// TwinCAT 3 PLC project Untitled1
// ProgramVersion: 3.1.4020.2
// libraries:
//   Tc2_SerialCom, * (Beckhoff Automation GmbH)
//   Tc2_SMS, * (Beckhoff Automation GmbH)
//   Tc2_Standard, * (Beckhoff Automation GmbH)
//   Tc2_System, * (Beckhoff Automation GmbH)
//   Tc2_Utilities, * (Beckhoff Automation GmbH)
//   Tc3_Module, * (Beckhoff Automation GmbH)
//   VisuDialogs, * (System)
// project tree:
//   / FAST_Serial.TcTTO, GlobalTextList.TcGTLO, PlcTask.TcTTO, Visualization Manager.TcVMO (not stored)
//   GVLs/ GVL.TcGVL
//   POUs/ KL6001_Serial.TcPOU, MAIN.TcPOU
//   VISUs/ Visualization.TcVIS
// real-time tasks:
//   TASK PlcTask: cycle T#10ms, priority 20, ADS port 350
//   TASK FAST_Serial: cycle T#1ms, priority 1, ADS port 351
// I/O:
//   DEVICE Device 3 (EtherCAT), AmsNetId 10.123.66.28.4.1
//     Box 1 (BK1150)
// variable links:
//   Untitled1/Untitled1 Instance <-> Device 3 (EtherCAT)/Box 1 (BK1150)
//     PlcTask Inputs/GVL.COMin_EL60xx/D[{0..4}] <-> Term 2 (KL6001-S)/Channel 1/Data In {0..4}  (5 links)
//     PlcTask Inputs/GVL.COMin_EL60xx/Status <-> Term 2 (KL6001-S)/Channel 1/State
//     PlcTask Outputs/GVL.COMout_EL60xx/Ctrl <-> Term 2 (KL6001-S)/Channel 1/Ctrl
//     PlcTask Outputs/GVL.COMout_EL60xx/D[{0..4}] <-> Term 2 (KL6001-S)/Channel 1/Data Out {0..4}  (5 links)

CONFIGURATION Untitled1
    RESOURCE PLC ON TwinCAT3
        TASK FAST_Serial(INTERVAL := T#1ms, PRIORITY := 1);
        TASK PlcTask(INTERVAL := T#10ms, PRIORITY := 20);
        PROGRAM KL6001_Serial WITH FAST_Serial : KL6001_Serial;
        PROGRAM MAIN WITH PlcTask : MAIN;
    END_RESOURCE
END_CONFIGURATION

// ---- GVLs/GVL.TcGVL

VAR_GLOBAL
	COMin_EL60xx	AT %I* 	: KL6InData5B;	(* linked to the EL60xx in the TwinCAT System Manager *)
	COMout_EL60xx	AT %Q*	: KL6OutData5B;	(* linked to the EL60xx in the TwinCAT System Manager *)
	RxBuffer: ComBuffer;						(* Receive data buffer; used with all receive function blocks *)
	TxBuffer: ComBuffer;						(* Transmit data buffer; used with all receive function blocks *)
END_VAR

// ---- POUs/KL6001_Serial.TcPOU
PROGRAM KL6001_Serial
VAR
	COMportControl: SerialLineControl;
	COMportControlError: BOOL;
	COMportControlErrorID: ComError_t;
END_VAR

(*==================================================================
	Background communication with KL6001 terminal
	The SerialLineControl function block is supposed to be called in every PLC cycle.
	It communicates with the serial line hardware device and transmits or receives data.
	The SerialLineControl can be called in the standard task or in a separate fast task as well.
	A fast separate task will be necessary at high baud rates or 
	with KL6001 terminals which have a small process image (3 or 5 data bytes only)
*)

(*
COMportControl(
	Mode:= SERIALLINEMODE_KL6_5B_STANDARD,
	pComIn:= ADR(COMin_EL60xx),			(* I/O data; see global variables *)
	pComOut:= ADR(COMout_EL60xx),		(* I/O data; see global variables *)
	SizeComIn:= SIZEOF(COMin_EL60xx),	(* I/O data; see global variables *)
	TxBuffer:= TxBuffer,				(* transmit buffer; see global variables *)
	RxBuffer:= RxBuffer,				(* receive buffer; see global variables *)
	Error=> COMportControlError,
	ErrorID=> COMportControlErrorID );
	
	*)

END_PROGRAM

// ---- POUs/MAIN.TcPOU
PROGRAM MAIN
VAR
	fbSerialInit: SerialLineControlADS;
	fbSendSMS 	: SendSMS;	
	
	//Variable to be changed
	stSerialCfg : ComSerialConfig := (ComPort := 3, BaudRate := 9600);
	sPhoneNo	: STRING := '83383193';
	sText 		: STRING := 'Test';
	
	bSerial		: BOOL := TRUE;
	bSendSMS 	: BOOL;
	bPortOpened	: BOOL;
	
	sRawReceive	: T_MAXSTRING;
	ptr 		: POINTER TO BYTE;
	i 			: INT;
	
	//SendATCommand
	bSend		: BOOL;
	sATCommand	: T_MAXSTRING := 'AT+CMGL="REC UNREAD"';
	sReceive 	: T_MAXSTRING;
	sendStr 	: SendSTring;
	sendByt		: SendByte;
	receiveStr	: ReceiveString;
	arrStr 		: ARRAY[0..20] OF STRING;
	j			: INT := 0;
	
	alarm 		: BOOL;
	alarm2		: BOOL;
END_VAR

(*------ Open the serial port ------*)
fbSerialInit(
	Connect:= bSerial, 
	SerialCfg:= stSerialCfg,
	Timeout:= , 
	TxBuffer:= TxBuffer, 
	RxBuffer:= RxBuffer, 
	PortOpened=> bPortOpened);

(*------ Send SMS ------*)
fbSendSMS(
	Send:= bSendSMS, 
	Number:= sPhoneNo, 
	Text:= sText, 
	Busy=> , 
	Error=> , 
	RXbuffer:= RxBuffer, 
	TXbuffer:= TxBuffer);

IF NOT fbSendSMS.Busy AND fbSendSMS.Error = 0 THEN
	fbSendSMS.Send := FALSE;
	bSendSMS := FALSE;
END_IF

(*------ Convert byte array to string ------*)
ptr:=ADR(sRawReceive);
FOR i:=0 TO 254 DO
	ptr^ := RxBuffer.Buffer[i];
	ptr:=ptr+1;
END_FOR

(*------ Receive SMS ------*)
ReceiveSMS();

ACTION ReceiveSMS:
(*------ Send AT Command ------*)
IF bSend THEN
	sendStr(SendString:= sATCommand, Busy=> , Error=> , TXbuffer:= TxBuffer);
	sendByt(SendByte:=13, Busy=> , Error=> , TxBuffer:= TxBuffer);
	bSend := FALSE;
END_IF

(*------ Filter the message received ------*)
receiveStr(
	Prefix:= 'Alert:', 
	Suffix:= 'Over.', 
	Timeout:= T#5S, 
	Reset:= , 
	StringReceived=> , 
	Busy=> , 
	Error=> , 
	RxTimeout=> , 
	ReceivedString:= sReceive, 
	RXbuffer:= RxBuffer);

(*------ Store the filtered message in string array ------*)
IF sReceive <> '' THEN
	IF j < 20 THEN
		arrStr[j] := sReceive;
		j := j+1;
	ELSE
		j := 0;
	END_IF
END_IF

(*------ Compare the message received with the message sent ------*)
IF sReceive = 'Alert: This is an announcement. Over.' THEN
	alarm := FALSE;
	sReceive := '';
ELSIF sReceive = 'Alert: This is the 2nd announcement. Over.' THEN
	alarm2 := FALSE;
	sReceive := '';
ELSE 
	sReceive := '';
END_IF
END_ACTION

END_PROGRAM

// ---- GlobalTextList.TcGTLO
TEXTLIST GlobalTextList
  5 = '%d'
  6 = '%s'
  13 = '(Data size: 8, Stop bit: 1, No parity)'
  9 = 'Alarm 1'
  10 = 'Alarm 2'
  2 = 'Baud Rate'
  1 = 'Com Port'
  8 = 'Filtered value'
  12 = 'Raw data received'
  4 = 'Received'
  11 = 'Received SMS'
  3 = 'Send'
  7 = 'Send AT Command'
  0 = 'Serial Connect'
END_TEXTLIST

// ---- VISUs/Visualization.TcVIS
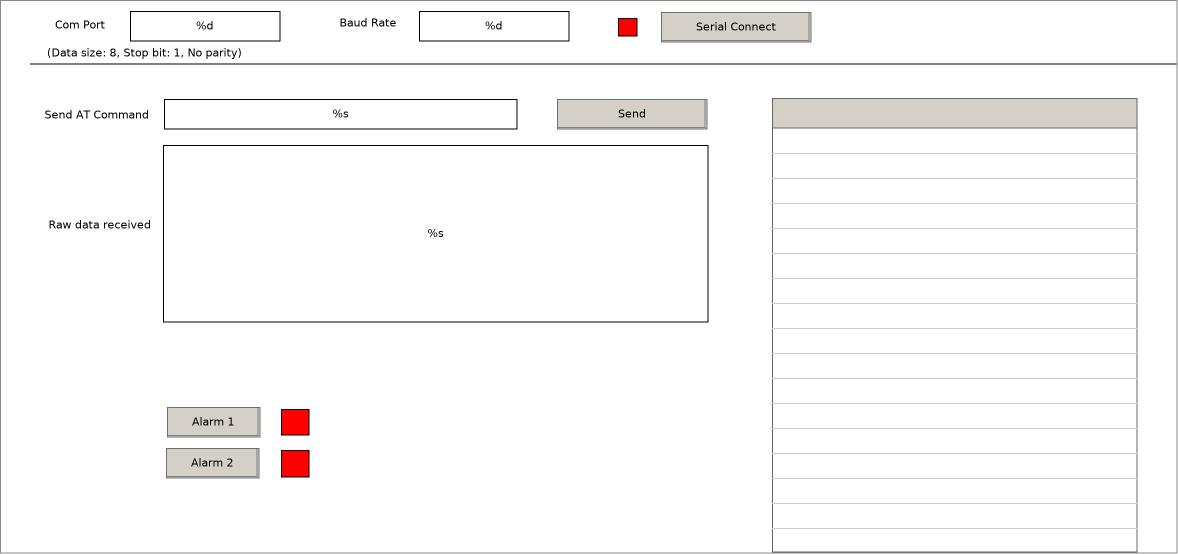
VISUALIZATION Visualization  // 1178x554
    Button (661,12 150x30), "Serial Connect"
        toggle MAIN.bSerial
    Rectangle (130,11 150x30), "%d", text variable: MAIN.stSerialCfg.ComPort
        OnMouseDown: write the text variable via Default
    Rectangle (419,11 150x30), "%d", text variable: MAIN.stSerialCfg.Baudrate
        OnMouseDown: write the text variable via Default
    Label (5,10 150x30), "Com Port"
    Label (293,8 150x30), "Baud Rate"
    Rectangle (164,99 353x30), "%s", text variable: MAIN.sATCommand
        OnMouseDown: write the text variable via Default
    Label (22,100 150x30), "Send AT Command"
    Label (25,210 150x30), "Raw data received"
    Rectangle (163,145 545x177), "%s", text variable: MAIN.sRawReceive
    Button (557,99 150x30), "Send"
        toggle MAIN.bSend
    Rectangle (618,18 19x18), colour toggle: MAIN.bPortOpened
    Rectangle (281,409 28x26), colour toggle: MAIN.alarm
    Rectangle (281,450 28x27), colour toggle: MAIN.alarm2
    Button (167,407 93x30), "Alarm 1"
        toggle MAIN.alarm
    Button (166,448 93x30), "Alarm 2"
        toggle MAIN.alarm2
    Table (772,98 365x454), data array: MAIN.arrStr
        p3854506369: MAIN.arrStr[INDEX]
        p2232123230: Received SMS
    Line (1176,64) (30,64)
    Label (15,38 259x30), "(Data size: 8, Stop bit: 1, No parity)"
END_VISUALIZATION
